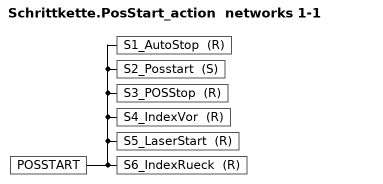
[picture p24: Schrittkette.PosStart_action (FBD) networks 1-1]
_FBD_ (* Function Block Diagram *)
NETWORK 1
	POSSTART => R S1_AutoStop, S S2_Posstart, R S3_POSStop, R S4_IndexVor, R S5_LaserStart, R S6_IndexRueck
_END_FBD_
(* the same logic as Structured Text *)
(* Network 1 *)
IF POSSTART THEN S1_AutoStop := FALSE; S2_Posstart := TRUE; S3_POSStop := FALSE; S4_IndexVor := FALSE; S5_LaserStart := FALSE; S6_IndexRueck := FALSE; END_IF;
END_ACTION

ACTION PosStop_action:
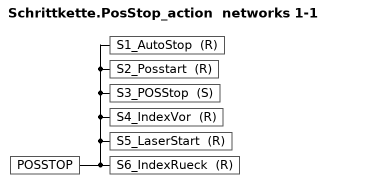
_FBD_ (* Function Block Diagram *)
NETWORK 1
	POSSTOP => R S1_AutoStop, R S2_Posstart, S S3_POSStop, R S4_IndexVor, R S5_LaserStart, R S6_IndexRueck
_END_FBD_
(* the same logic as Structured Text *)
(* Network 1 *)
IF POSSTOP THEN S1_AutoStop := FALSE; S2_Posstart := FALSE; S3_POSStop := TRUE; S4_IndexVor := FALSE; S5_LaserStart := FALSE; S6_IndexRueck := FALSE; END_IF;
END_ACTION

ACTION IndexVor_action:
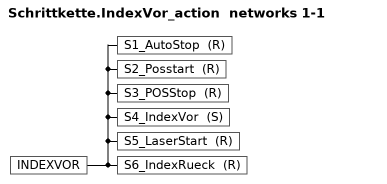
_FBD_ (* Function Block Diagram *)
NETWORK 1
	INDEXVOR => R S1_AutoStop, R S2_Posstart, R S3_POSStop, S S4_IndexVor, R S5_LaserStart, R S6_IndexRueck
_END_FBD_
(* the same logic as Structured Text *)
(* Network 1 *)
IF INDEXVOR THEN S1_AutoStop := FALSE; S2_Posstart := FALSE; S3_POSStop := FALSE; S4_IndexVor := TRUE; S5_LaserStart := FALSE; S6_IndexRueck := FALSE; END_IF;
END_ACTION

ACTION LaserStart_action:
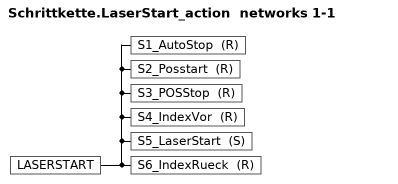
_FBD_ (* Function Block Diagram *)
NETWORK 1
	LASERSTART => R S1_AutoStop, R S2_Posstart, R S3_POSStop, R S4_IndexVor, S S5_LaserStart, R S6_IndexRueck
_END_FBD_
(* the same logic as Structured Text *)
(* Network 1 *)
IF LASERSTART THEN S1_AutoStop := FALSE; S2_Posstart := FALSE; S3_POSStop := FALSE; S4_IndexVor := FALSE; S5_LaserStart := TRUE; S6_IndexRueck := FALSE; END_IF;
END_ACTION

ACTION IndexRueck_action:
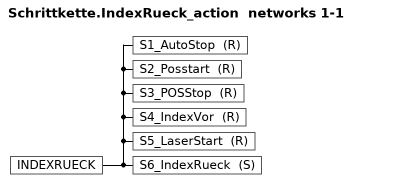
_FBD_ (* Function Block Diagram *)
NETWORK 1
	INDEXRUECK => R S1_AutoStop, R S2_Posstart, R S3_POSStop, R S4_IndexVor, R S5_LaserStart, S S6_IndexRueck
_END_FBD_
(* the same logic as Structured Text *)
(* Network 1 *)
IF INDEXRUECK THEN S1_AutoStop := FALSE; S2_Posstart := FALSE; S3_POSStop := FALSE; S4_IndexVor := FALSE; S5_LaserStart := FALSE; S6_IndexRueck := TRUE; END_IF;
END_ACTION

TRANSITION Trans2:
_FBD_ (* Function Block Diagram *)
NETWORK 1
	AND(RegMarkierung[ZeigerReg].1, NOT RegMarkierung[ZeigerReg].2, S_MAutoStart)
_END_FBD_
END_TRANSITION

TRANSITION Trans8:
_FBD_ (* Function Block Diagram *)
NETWORK 1
	AND(NOT PosErreicht, S_MAutoStop)
_END_FBD_
END_TRANSITION

TRANSITION Trans4:
_FBD_ (* Function Block Diagram *)
NETWORK 1
	AND(TON_IIndexVor.Q, NOT Sammelstoerung)
_END_FBD_
END_TRANSITION

TRANSITION Trans9:
_FBD_ (* Function Block Diagram *)
NETWORK 1
	Sammelstoerung
_END_FBD_
(* the same logic as Structured Text *)
(* Network 1 *)
Trans9 := Sammelstoerung;
END_TRANSITION

TRANSITION Trans6:
_FBD_ (* Function Block Diagram *)
NETWORK 1
	AND(NOT S_MAutoStart, IINI_IndexRueck)
_END_FBD_
END_TRANSITION

TRANSITION Trans7:
_FBD_ (* Function Block Diagram *)
NETWORK 1
	AND(S_MAutoStart, IINI_IndexRueck)
_END_FBD_
END_TRANSITION
END_PROGRAM
